{attribute 'linkalways'} 
{attribute 'no_explicit_call' := 'This FB is a CLASS and must be accessed using methods or properties'}
{attribute 'enable_dynamic_creation'}
FUNCTION_BLOCK Node_F_VN_AppendToContainer_TcVnVector2_INT EXTENDS VisionNode
VAR
    aElement : _TcVnVector2_INT;
    ipContainer : _ITcVnContainer;
    hrPrev : _HRESULT(S_OK);
	hresult : _HRESULT(S_OK);
END_VAR

METHOD PUBLIC  Clone : I_Node
VAR
	pNode : POINTER TO Node_F_VN_AppendToContainer_TcVnVector2_INT;
END_VAR
pNode := __NEW(Node_F_VN_AppendToContainer_TcVnVector2_INT);
Clone := pNode^;
END_METHOD

METHOD FB_init : BOOL
VAR_INPUT
	bInitRetains : BOOL; // if TRUE, the retain variables are initialized (warm start / cold start)
	bInCopyCode : BOOL;  // if TRUE, the instance afterwards gets moved into the copy code (online change)
END_VAR
AddInput('aElement', aElement);
AddInput('ipContainer', ipContainer);
AddInput('hrPrev', hrPrev);
AddOutput('ipContainer', ipContainer);
AddOutput('hresult',hresult);
END_METHOD

METHOD PROTECTED OnExecute
hresult.Value := F_VN_AppendToContainer_TcVnVector2_INT(
    aElement := aElement.Value,
	ipContainer := ipContainer.Value,
	hrPrev:= hrPrev.Value);
END_METHOD

METHOD PUBLIC PreExecutionCheck
VAR_INPUT
	Check : I_PreExecutionChecks;
END_VAR
Check.IsTrue(ipContainer.IsValid, 'ipContainer must be a valid container');
Check.IsTrue(ipContainer.IsType(TC_GLOBAL_CONST_LIST.ContainerType_Vector_TcVnVector2_INT), 'ipContainer contains incorrect type');
END_METHOD

END_FUNCTION_BLOCK

(* stored: Version 1.1.0.1, ProductVersion 3.1.4026.13
   POU Node_F_VN_AppendToContainer_TcVnVector2_INT: Id {207d187b-da09-4b67-9c09-a2e734da284b}, SpecialFunc None
   Folder Constructor: Id {ab8a9f63-2b87-4775-a578-12604b83e21a}
   Method Clone: Id {dcaf24c5-d9e7-4f33-b870-29c9c8e855c5}
   Method FB_init: Id {63d1e4ce-69c9-42f0-8bf1-0604068ed8a1}
   Method OnExecute: Id {05b5e95e-e2d3-49d8-adce-cdf07af29c04}
   Method PreExecutionCheck: Id {a0a78ebe-1193-4813-9dc0-025459fc631c} *)
